Staubli VAL3: TestPositionCal.pgx

program TestPositionCal()
begin
  call DeplacementInit()

  call Deplacementpion(0,1)
  call Deplacementpion(31,30)
end
